FUNCTION_BLOCK TEST_CONDITION (* Service Interface Function Block Type *)
  PACKAGE eclipse4diac::utils;
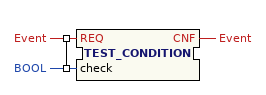
  EVENT_INPUT
    REQ WITH check; (* Request Test *)
  END_EVENT
  EVENT_OUTPUT
    CNF; (* Test finished *)
  END_EVENT
  VAR_INPUT
    check : BOOL; (* Test fails if check == 0, passes otherwise *)
  END_VAR
END_FUNCTION_BLOCK
